// TIA Portal V19 export
FUNCTION "FC_FW_Auftrag_Step1_NB" : Void   // FC181, LAD
TITLE = Schritt CM01/CMD02 -> CM03
{ S7_Optimized_Access := 'TRUE' }
// Ältesten Warenträger in CM01/CM02 suchen und nach CM03 transportieren
// stored: AutoNumber false, SetENOAutomatically false
   VAR_INPUT
      Frg_Schritt : Bool;
   END_VAR
   VAR_OUTPUT
      nextStep : Bool;
      startStep : Bool;
      parkStep : Bool;
   END_VAR
   VAR_IN_OUT
      Quelle : Int;
      Ziel : Int;
      Positionen : Array[1..30] of "UDT_Auftrag_Pos";
   END_VAR
   VAR_TEMP
      Sperre_Kurz_li : Bool;
      Sperre_Kurz_re : Bool;
      Sperre_Lang : Bool;
      Vorzug : Bool;
      Befehl_ok : Bool;
      tmpQuelle : Int;
      Oldest : Real;
   END_VAR
BEGIN

REGION Network 1 (SCL): Initialisieren
   IF (#Quelle <> 0) AND (#Ziel <> 0) THEN
       #nextStep := #Positionen[#Quelle].Sperre;
       #startStep := NOT #nextStep;
       #Quelle := 0;
       #Ziel := 0;
       RETURN;
   END_IF;

   #Quelle := 0;
   #Ziel := 0;
   #nextStep := FALSE;
   #startStep := FALSE;

   IF NOT #Frg_Schritt THEN
       #nextStep := TRUE;
       RETURN;
   END_IF;
END_REGION

REGION Network 2 (SCL): Positionen sperren
   //Groß links nicht möglich
   #Positionen[3].CheckSperre := #Positionen[9].Sperre;
   #Positionen[15].CheckSperre := #Positionen[9].Sperre;

   //Groß rechts nicht möglich
   #Positionen[4].CheckSperre := #Positionen[10].Sperre;
   #Positionen[16].CheckSperre := #Positionen[10].Sperre;

   //kein Platz für Kurz links in CM03
   #Sperre_Kurz_li := #Positionen[7].Sperre AND #Positionen[11].Sperre;

   //kein Platz für Kurz rechts in CM03
   #Sperre_Kurz_re := #Positionen[8].Sperre AND #Positionen[12].Sperre;

   //kein Platz für Lang in CM03
   #Sperre_Lang := (#Positionen[7].Sperre OR #Positionen[8].Sperre) AND (#Positionen[11].Sperre OR #Positionen[12].Sperre);

   //Lang in P1 oder
   //kein Platz auf rechter Seite
   //-> P2 sperren
   #Positionen[2].CheckSperre := #Sperre_Kurz_re OR (#Positionen[1].Wt_Typ = "WT_Typ_LS");

   //Lang in P1 und kein Platz für Lang oder
   //kein Platz auf linker Seite
   //-> P1 sperren
   #Positionen[1].CheckSperre := #Sperre_Kurz_li OR ((#Positionen[1].Wt_Typ = "WT_Typ_LS") AND #Sperre_Lang);

   //Lang in P5 oder
   //kein Platz auf rechter Seite
   //-> P6 sperren
   #Positionen[6].CheckSperre := #Sperre_Kurz_re OR (#Positionen[5].Wt_Typ = "WT_Typ_LS");

   //Lang in P5 und kein Platz für Lang oder
   //kein Platz auf linker Seite
   //-> P5 sperren
   #Positionen[5].CheckSperre := #Sperre_Kurz_li OR ((#Positionen[5].Wt_Typ = "WT_Typ_LS") AND #Sperre_Lang);

   //Lang in P13 oder
   //kein Platz auf rechter Seite
   //-> P14 sperren
   #Positionen[14].CheckSperre := #Sperre_Kurz_re OR (#Positionen[13].Wt_Typ = "WT_Typ_LS");

   //Lang in P13 und kein Platz für Lang oder
   //kein Platz auf linker Seite
   //-> P13 sperren
   #Positionen[13].CheckSperre := #Sperre_Kurz_li OR ((#Positionen[13].Wt_Typ = "WT_Typ_LS") AND #Sperre_Lang);

   //Lang in P17 oder
   //kein Platz auf rechter Seite
   //-> P18 sperren
   #Positionen[18].CheckSperre := #Sperre_Kurz_re OR (#Positionen[17].Wt_Typ = "WT_Typ_LS");

   //Lang in P17 und kein Platz für Lang oder
   //kein Platz auf linker Seite
   //-> P17 sperren
   #Positionen[17].CheckSperre := #Sperre_Kurz_li OR ((#Positionen[17].Wt_Typ = "WT_Typ_LS") AND #Sperre_Lang);
END_REGION

REGION Network 3 (SCL): Ältesten WT suchen
   //
   #Oldest := 0;
   #tmpQuelle := 0;

   //CM01
   "FC_FW_Auftrag_Suche"(Pos1 := 1,
                         Pos2 := 6,
                         Positionen := #Positionen,
                         Quelle := #tmpQuelle,
                         Oldest := #Oldest);

   //CM02
   "FC_FW_Auftrag_Suche"(Pos1 := 13,
                         Pos2 := 18,
                         Positionen := #Positionen,
                         Quelle := #tmpQuelle,
                         Oldest := #Oldest);
END_REGION

REGION Network 4 (SCL): Auswertung
   IF #tmpQuelle = 0 THEN
       //kein WT
       #nextStep := TRUE;
       RETURN;
   END_IF;

   IF ("DI_FW_1".ZST.POSITION_li <= 6) AND (#tmpQuelle <= 6) THEN
       //schieben wenn über Quelle CM01
       "FC_FW_Auftrag_Befehl"(inQuelle := 7,
                              inZiel := 0,
                              Befehl_ok => #Befehl_ok,
                              outQuelle => #Quelle,
                              outZiel => #Ziel);

       #nextStep := NOT #Befehl_ok;
       RETURN;
   END_IF;

   IF ("DI_FW_1".ZST.POSITION_li >= 13) AND ("DI_FW_1".ZST.POSITION_li <= 18) AND (#tmpQuelle >= 13) THEN
       //schieben wenn über Quelle CM02
       "FC_FW_Auftrag_Befehl"(inQuelle := 11,
                              inZiel := 0,
                              Befehl_ok => #Befehl_ok,
                              outQuelle => #Quelle,
                              outZiel => #Ziel);

       #nextStep := NOT #Befehl_ok;
       RETURN;
   END_IF;

   IF NOT #Positionen[#tmpQuelle].Fertig THEN
       #parkStep := TRUE;
       RETURN;
   END_IF;

   IF (#tmpQuelle = 3) OR (#tmpQuelle = 15) THEN
       //Gross links
       IF NOT #Positionen[9].Sperre THEN
           "FC_FW_Auftrag_Befehl"(inQuelle := #tmpQuelle,
                                  inZiel := 9,
                                  Befehl_ok => #Befehl_ok,
                                  outQuelle => #Quelle,
                                  outZiel => #Ziel);

           #nextStep := NOT #Befehl_ok;
       ELSE
           #nextStep := TRUE;
       END_IF;
       RETURN;
   END_IF;

   IF (#tmpQuelle = 4) OR (#tmpQuelle = 16) THEN
       //Gross rechts
       IF NOT #Positionen[10].Sperre THEN
           "FC_FW_Auftrag_Befehl"(inQuelle := #tmpQuelle,
                                  inZiel := 10,
                                  Befehl_ok => #Befehl_ok,
                                  outQuelle => #Quelle,
                                  outZiel => #Ziel);

           #nextStep := NOT #Befehl_ok;
       ELSE
           #nextStep := TRUE;
       END_IF;
       RETURN;
   END_IF;

   IF (#Positionen[#tmpQuelle].Wt_Typ = "WT_Typ_LS") AND ((#tmpQuelle = 1) OR (#tmpQuelle = 5) OR (#tmpQuelle = 13) OR (#tmpQuelle = 17)) THEN
       //Lang
       IF NOT #Positionen[7].Sperre AND NOT #Positionen[8].Sperre THEN
           "FC_FW_Auftrag_Befehl"(inQuelle := #tmpQuelle,
                                  inZiel := 7,
                                  Befehl_ok => #Befehl_ok,
                                  outQuelle => #Quelle,
                                  outZiel => #Ziel);

           #nextStep := NOT #Befehl_ok;
       ELSIF NOT #Positionen[11].Sperre AND NOT #Positionen[12].Sperre THEN
           "FC_FW_Auftrag_Befehl"(inQuelle := #tmpQuelle,
                                  inZiel := 11,
                                  Befehl_ok => #Befehl_ok,
                                  outQuelle => #Quelle,
                                  outZiel => #Ziel);

           #nextStep := NOT #Befehl_ok;
       ELSE
           #nextStep := TRUE;
       END_IF;
       RETURN;
   END_IF;

   IF (#tmpQuelle = 1) OR (#tmpQuelle = 5) OR (#tmpQuelle = 13) OR (#tmpQuelle = 17) THEN
       //Kurz links
       #Vorzug := NOT #Positionen[7].Sperre AND NOT #Positionen[8].Sperre AND NOT #Positionen[11].Sperre AND #Positionen[12].Sperre;

       IF NOT #Positionen[7].Sperre AND NOT #Vorzug THEN
           "FC_FW_Auftrag_Befehl"(inQuelle := #tmpQuelle,
                                  inZiel := 7,
                                  Befehl_ok => #Befehl_ok,
                                  outQuelle => #Quelle,
                                  outZiel => #Ziel);

           #nextStep := NOT #Befehl_ok;
       ELSIF NOT #Positionen[11].Sperre THEN
           "FC_FW_Auftrag_Befehl"(inQuelle := #tmpQuelle,
                                  inZiel := 11,
                                  Befehl_ok => #Befehl_ok,
                                  outQuelle => #Quelle,
                                  outZiel => #Ziel);

           #nextStep := NOT #Befehl_ok;
       ELSE
           #nextStep := TRUE;
       END_IF;
       RETURN;
   END_IF;

   IF (#tmpQuelle = 2) OR (#tmpQuelle = 6) OR (#tmpQuelle = 14) OR (#tmpQuelle = 18) THEN
       //Kurz rechts
       #Vorzug := NOT #Positionen[7].Sperre AND NOT #Positionen[8].Sperre AND #Positionen[11].Sperre AND NOT #Positionen[12].Sperre;

       IF NOT #Positionen[8].Sperre AND NOT #Vorzug THEN
           "FC_FW_Auftrag_Befehl"(inQuelle := #tmpQuelle,
                                  inZiel := 8,
                                  Befehl_ok => #Befehl_ok,
                                  outQuelle => #Quelle,
                                  outZiel => #Ziel);

           #nextStep := NOT #Befehl_ok;
       ELSIF NOT #Positionen[12].Sperre THEN
           "FC_FW_Auftrag_Befehl"(inQuelle := #tmpQuelle,
                                  inZiel := 12,
                                  Befehl_ok => #Befehl_ok,
                                  outQuelle => #Quelle,
                                  outZiel => #Ziel);

           #nextStep := NOT #Befehl_ok;
       ELSE
           #nextStep := TRUE;
       END_IF;
       RETURN;
   END_IF;

   //?
   #nextStep := TRUE;
END_REGION
END_FUNCTION
